LIN {X 0,Y 87.309,Z 428.793,A -85,B 0,C 180,E1 -31155.247,E2 -31155.247} C_VEL
LIN {X 0,Y 84.983,Z 444.184,A -85,B 0,C 180,E1 -31155.675,E2 -31155.675} C_VEL
LIN {X 0,Y 81.797,Z 456.363,A -85,B 0,C 180,E1 -31156.1,E2 -31156.1} C_VEL
LIN {X 0,Y 77.075,Z 468.971,A -85,B 0,C 180,E1 -31156.763,E2 -31156.763} C_VEL
LIN {X 0,Y 71.103,Z 481.086,A -85,B 0,C 180,E1 -31157.93,E2 -31157.93} C_VEL
LIN {X 0,Y 64.22,Z 491.93,A -85,B 0,C 180,E1 -31159.258,E2 -31159.258} C_VEL
LIN {X 0,Y 56.506,Z 501.788,A -85,B 0,C 180,E1 -31161.104,E2 -31161.104} C_VEL
LIN {X 0,Y 48.03,Z 510.744,A -85,B 0,C 180,E1 -31163.844,E2 -31163.844} C_VEL
LIN {X 0,Y 38.005,Z 519.486,A -85,B 0,C 180,E1 -31168.532,E2 -31168.532} C_VEL
LIN {X 0,Y 28.402,Z 526.446,A -85,B 0,C 180,E1 -31176.447,E2 -31176.447} C_VEL
LIN {X 0,Y 18.368,Z 532.854,A -85,B 0,C 180,E1 -31194.952,E2 -31194.952} C_VEL
LIN {X 0,Y 12.799,Z 537.085,A -85,B 0,C 180,E1 -31229.972,E2 -31229.972} C_VEL
LIN {X 0,Y 13.376,Z 539.534,A -85,B 0,C 180,E1 -31266.297,E2 -31266.297} C_VEL
LIN {X 0,Y 14.628,Z 540.518,A -85,B 0,C 180,E1 -31281.327,E2 -31281.327} C_VEL
LIN {X 0,Y 17.08,Z 541.764,A -85,B 0,C 180,E1 -31303.72,E2 -31303.72} C_VEL
LIN {X 0,Y 21.387,Z 542.764,A -85,B 0,C 180,E1 -31319.101,E2 -31319.101} C_VEL
LIN {X 0,Y 24.961,Z 543.203,A -85,B 0,C 180,E1 -31323.348,E2 -31323.348} C_VEL
LIN {X 0,Y 28.212,Z 543.581,A -85,B 0,C 180,E1 -31324.99,E2 -31324.99} C_VEL
LIN {X 0,Y 28.293,Z 543.61,A -85,B 0,C 180,E1 -31326.606,E2 -31326.606} C_VEL
LIN {X 0,Y 21.468,Z 542.921,A -85,B 0,C 180,E1 -31330.944,E2 -31330.944} C_VEL
LIN {X 0,Y 14.863,Z 541.806,A -85,B 0,C 180,E1 -31339.038,E2 -31339.038} C_VEL
LIN {X 0,Y 8.939,Z 540.292,A -85,B 0,C 180,E1 -31358.233,E2 -31358.233} C_VEL
LIN {X 0,Y 5.916,Z 538.356,A -85,B 0,C 180,E1 -31410.062,E2 -31410.062} C_VEL
LIN {X 0,Y 11.683,Z 534.477,A -85,B 0,C 180,E1 -31474.535,E2 -31474.535} C_VEL
LIN {X 0,Y 21.407,Z 529.417,A -85,B 0,C 180,E1 -31490.138,E2 -31490.138} C_VEL
LIN {X 0,Y 31.722,Z 523.05,A -85,B 0,C 180,E1 -31495.68,E2 -31495.68} C_VEL
LIN {X 0,Y 42.181,Z 515.009,A -85,B 0,C 180,E1 -31498.922,E2 -31498.922} C_VEL
LIN {X 0,Y 50.96,Z 506.826,A -85,B 0,C 180,E1 -31500.399,E2 -31500.399} C_VEL
LIN {X 0,Y 59.765,Z 496.812,A -85,B 0,C 180,E1 -31501.523,E2 -31501.523} C_VEL
LIN {X 0,Y 65.062,Z 489.529,A -85,B 0,C 180,E1 -31502.192,E2 -31502.192} C_VEL
LIN {X 0,Y 71.232,Z 479.507,A -85,B 0,C 180,E1 -31502.495,E2 -31502.495} C_VEL
LIN {X 0,Y 75.65,Z 470.698,A -85,B 0,C 180,E1 -31502.845,E2 -31502.845} C_VEL
LIN {X 0,Y 80.532,Z 458.191,A -85,B 0,C 180,E1 -31503.143,E2 -31503.143} C_VEL
LIN {X 0,Y 84.018,Z 445.57,A -85,B 0,C 180,E1 -31503.379,E2 -31503.379} C_VEL
LIN {X 0,Y 86.073,Z 433.411,A -85,B 0,C 180,E1 -31503.578,E2 -31503.578} C_VEL
LIN {X 0,Y 86.061,Z 432.828,A -85,B 0,C 180,E1 -31504.683,E2 -31504.683} C_VEL
LIN {X 0,Y 86.014,Z 433.074,A -85,B 0,C 180,E1 -31509.404,E2 -31509.404} C_VEL
LIN {X 0,Y 86.019,Z 433.677,A -85,B 0,C 180,E1 -31510.601,E2 -31510.601} C_VEL
LIN {X 0,Y 83.839,Z 446.118,A -85,B 0,C 180,E1 -31510.908,E2 -31510.908} C_VEL
LIN {X 0,Y 80.105,Z 459.224,A -85,B 0,C 180,E1 -31511.166,E2 -31511.166} C_VEL
LIN {X 0,Y 75.337,Z 471.184,A -85,B 0,C 180,E1 -31511.593,E2 -31511.593} C_VEL
LIN {X 0,Y 69.255,Z 482.771,A -85,B 0,C 180,E1 -31512.358,E2 -31512.358} C_VEL
LIN {X 0,Y 62.191,Z 493.384,A -85,B 0,C 180,E1 -31513.061,E2 -31513.061} C_VEL
LIN {X 0,Y 54.347,Z 502.983,A -85,B 0,C 180,E1 -31514.071,E2 -31514.071} C_VEL
LIN {X 0,Y 45.615,Z 511.774,A -85,B 0,C 180,E1 -31515.618,E2 -31515.618} C_VEL
LIN {X 0,Y 35.158,Z 520.316,A -85,B 0,C 180,E1 -31518.251,E2 -31518.251} C_VEL
LIN {X 0,Y 24.834,Z 527.161,A -85,B 0,C 180,E1 -31523.072,E2 -31523.072} C_VEL
LIN {X 0,Y 13.135,Z 533.469,A -85,B 0,C 180,E1 -31536.574,E2 -31536.574} C_VEL
LIN {X 0,Y 5.505,Z 537.608,A -85,B 0,C 180,E1 -31589.934,E2 -31589.934} C_VEL
LIN {X 0,Y 7.925,Z 539.751,A -85,B 0,C 180,E1 -31652.379,E2 -31652.379} C_VEL
LIN {X 0,Y 20.201,Z 542.598,A -85,B 0,C 180,E1 -31680.005,E2 -31680.005} C_VEL
LIN {X 0,Y 24.961,Z 543.203,A -85,B 0,C 180,E1 -31683.348,E2 -31683.348} C_VEL
LIN {X 0,Y 26.686,Z 545.19,A -85,B 0,C 180,E1 -31684.27,E2 -31684.27} C_VEL
LIN {X 0,Y 26.686,Z 600,A -85,B 0,C 180,E1 -31684.27,E2 -31684.27} C_VEL
LIN {X 0,Y 26.686,Z 600,A -85,B 0,C 180,E1 -31684.27,E2 -31684.27}

QRS_NEXT_CUT()

QRS_NEXT()
QRS_HOME()

END
